KUKA KRL program: ResetaPallet.src, ResetaPallet.dat

--- ResetaPallet.src ---
&ACCESS RVO
&REL 3
&PARAM EDITMASK = *
DEF ResetaPallet( )
   ;precisa saber qual o pallet Atual
   ;atravez do pallet Atual o programa sabe qual mozaico est� selecionado

   ;FOLD RESETA PALLET
      ;StrPallet[PalletAtual].Livre=TRUE
      ;StrPallet[PalletAtual].ReceitaAtual=1
      StrPallet[PalletAtual].PlaceAtual=1
      StrPallet[PalletAtual].CamadaAtual=1
   ;ENDFOLD

END

--- ResetaPallet.dat ---
DEFDAT  ResetaPallet

ENDDAT
